DEVICE_TYPE _TCREST
  (* Standard: 61499-2 *)
  (* Version 0.1, 2017-00-09, hpea485, UOA *)
  RESOURCE rx_core : _Core0(RxChanId := 1)
  END_RESOURCE
  RESOURCE tx_core : _Core1(TxChanId := 1)
  END_RESOURCE
END_DEVICE_TYPE
